// TIA Portal V20 export
TYPE "typeSequenceControlNodeJobInterfaceCommands"
// stored: Namespace Unit1.Em1
   STRUCT
      reqAutoSplice { ExternalWritable := 'False'} : Bool;
   END_STRUCT;
END_TYPE
